FUNCTION_BLOCK Top
  (* Standard: 61499-2 *)
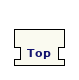
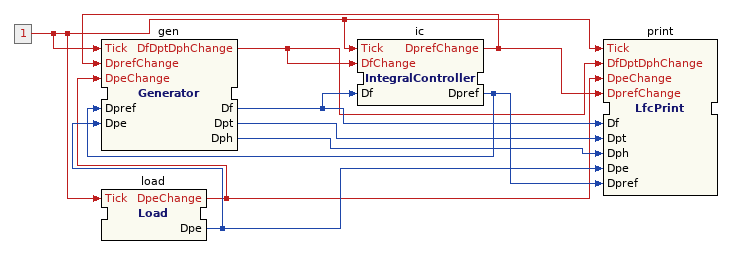
  FBS
    gen : Generator;
    ic : IntegralController;
    print : LfcPrint;
    load : Load;
  END_FBS
  EVENT_CONNECTIONS
    1 TO ic.Tick;
    1 TO gen.Tick;
    1 TO print.Tick;
    1 TO load.Tick;
    load.DpeChange TO print.DpeChange;
    gen.DfDptDphChange TO ic.DfChange;
    ic.DprefChange TO gen.DprefChange;
    load.DpeChange TO gen.DpeChange;
    gen.DfDptDphChange TO print.DfDptDphChange;
    ic.DprefChange TO print.DprefChange;
  END_CONNECTIONS
  DATA_CONNECTIONS
    gen.Df TO ic.Df;
    ic.Dpref TO gen.Dpref;
    load.Dpe TO gen.Dpe;
    gen.Df TO print.Df;
    gen.Dpt TO print.Dpt;
    gen.Dph TO print.Dph;
    ic.Dpref TO print.Dpref;
    load.Dpe TO print.Dpe;
  END_CONNECTIONS
END_FUNCTION_BLOCK
